// TIA Portal V20 export
VAR_GLOBAL   // PLC tag table "PLC tags"
END_VAR
